FUNCTION_BLOCK I_RPTO (* Primary or Rear Power Take off Output Shaft RPTO *)
  (* Standard: ISO 11783-7; Classification: PGN 65091; Function: Primary or Rear Power Take off Output Shaft RPTO; Description: Copyright (c) 2024 HR Agrartechnik GmbH This program and the accompanying materials are made available under the terms of the Eclipse Public License 2.0 which is available at https://www.eclipse.org/legal/epl-2.0/ SPDX-License-Identifier: EPL-2.0 Message that provides the measurement of the current primary or rear power take-off (PTO) output shaft parameters. https://docs.ms-muc-docs.de/projects/isobus-other-docs/de/latest/PGN/PGN_65091.html *)
  (* Version 1.0, 2024-07-09, Franz Höpfinger, HR Agrartechnik GmbH *)
  PACKAGE isobus::tecu;
  (* Documentation:
  Primary or Rear Power Take off Output Shaft RPTO
   TIMEOUT / IND Vertrag: TIMEOUT feuert ausschliesslich beim tatsaechlichen Eintreten eines Timeouts (Q_timeout wird true). Das Zuruecksetzen von Q_timeout auf false (Timeout vorbei) wird bewusst NICHT nochmal separat ueber TIMEOUT gemeldet, sondern kommt ueber IND - das feuert bei jedem Zyklus ohne aktiven Timeout und publiziert Q_timeout mit. Nachgeschaltete Bausteine, die auf das Ende eines Timeouts reagieren muessen, werten dafuer IND mit Q_timeout==false aus, nicht ein zweites TIMEOUT-Event.
  *)
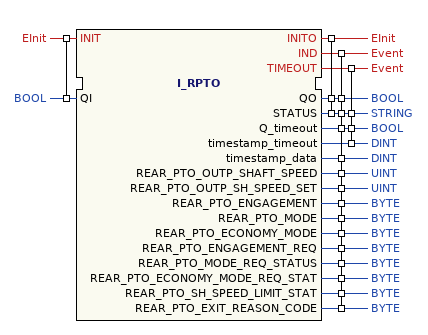
  EVENT_INPUT
    INIT : EInit WITH QI; (* Service Initialization *)
  END_EVENT
  EVENT_OUTPUT
    INITO : EInit WITH QO, STATUS; (* Initialization Confirm *)
    IND WITH QO, timestamp_data, STATUS, Q_timeout, REAR_PTO_OUTP_SHAFT_SPEED, REAR_PTO_OUTP_SH_SPEED_SET, REAR_PTO_ENGAGEMENT, REAR_PTO_MODE, REAR_PTO_ECONOMY_MODE, REAR_PTO_ENGAGEMENT_REQ, REAR_PTO_MODE_REQ_STATUS, REAR_PTO_ECONOMY_MODE_REQ_STAT, REAR_PTO_SH_SPEED_LIMIT_STAT, REAR_PTO_EXIT_REASON_CODE; (* Indication from Resource - feuert bei jedem Zyklus ohne aktiven Timeout und publiziert dabei auch den Reset von Q_timeout auf false. *)
    TIMEOUT WITH timestamp_timeout, STATUS, Q_timeout; (* Feuert ausschliesslich beim tatsaechlichen Eintreten eines Timeouts (Entry-Trigger). Das Zuruecksetzen von Q_timeout auf false wird NICHT hier, sondern ueber IND gemeldet. *)
  END_EVENT
  VAR_INPUT
    QI : BOOL; (* Event Input Qualifier *)
  END_VAR
  VAR_OUTPUT
    QO : BOOL; (* Event Output Qualifier *)
    STATUS : STRING;
    Q_timeout : BOOL;
    timestamp_timeout : DINT;
    timestamp_data : DINT;
    REAR_PTO_OUTP_SHAFT_SPEED : UINT := UINT#16#FFFF; (* Rear PTO output shaft speed (see Attributes for Details) *) {SET_ATTRIBUTE(SPN, 1883)} {SET_ATTRIBUTE(SPN_Name, 'Rear PTO output shaft speed')} {SET_ATTRIBUTE(SP_Position_In_PG, '1-2')} {SET_ATTRIBUTE(SP_Length, 16)} (* 16 bits *) {SET_ATTRIBUTE(Scaling, '0.125 1/min/bit')} {SET_ATTRIBUTE(Offset, )} {SET_ATTRIBUTE(Link, 'https://docs.ms-muc-docs.de/projects/isobus-other-docs/de/latest/PGN/PGN_65091.html#spn-1883-rear-pto-output-shaft-speed')}
    REAR_PTO_OUTP_SH_SPEED_SET : UINT := UINT#16#FFFF; (* Rear PTO Output Shaft Speed Set Point (see Attributes for Details) *) {SET_ATTRIBUTE(SPN, 1885)} {SET_ATTRIBUTE(SPN_Name, 'Rear PTO Output Shaft Speed Set Point')} {SET_ATTRIBUTE(SP_Position_In_PG, '3-4')} {SET_ATTRIBUTE(SP_Length, 16)} (* 16 bits *) {SET_ATTRIBUTE(Scaling, '0.125 1/min/bit')} {SET_ATTRIBUTE(Offset, )} {SET_ATTRIBUTE(Link, 'https://docs.ms-muc-docs.de/projects/isobus-other-docs/de/latest/PGN/PGN_65091.html#spn-1885-rear-pto-output-shaft-speed-set-point')}
    REAR_PTO_ENGAGEMENT : BYTE := BYTE#16#FF; (* Rear Power Take Off Engagement (see Attributes for Details) *) {SET_ATTRIBUTE(SPN, 2408)} {SET_ATTRIBUTE(SPN_Name, 'Rear Power Take Off Engagement')} {SET_ATTRIBUTE(SP_Position_In_PG, '5.7')} {SET_ATTRIBUTE(SP_Length, 2)} (* 2 bits *) {SET_ATTRIBUTE(Scaling, '4 states/2 bit')} {SET_ATTRIBUTE(Offset, )} {SET_ATTRIBUTE(Link, 'https://docs.ms-muc-docs.de/projects/isobus-other-docs/de/latest/PGN/PGN_65091.html#spn-2408-rear-power-take-off-engagement')}
    REAR_PTO_MODE : BYTE := BYTE#16#FF; (* Rear Power Take Off Mode (see Attributes for Details) *) {SET_ATTRIBUTE(SPN, 1890)} {SET_ATTRIBUTE(SPN_Name, 'Rear Power Take Off Mode')} {SET_ATTRIBUTE(SP_Position_In_PG, '5.5')} {SET_ATTRIBUTE(SP_Length, 2)} (* 2 bits *) {SET_ATTRIBUTE(Scaling, '4 states/2 bit')} {SET_ATTRIBUTE(Offset, )} {SET_ATTRIBUTE(Link, 'https://docs.ms-muc-docs.de/projects/isobus-other-docs/de/latest/PGN/PGN_65091.html#spn-1890-rear-power-take-off-mode')}
    REAR_PTO_ECONOMY_MODE : BYTE := BYTE#16#FF; (* Rear Power Take Off Economy Mode (see Attributes for Details) *) {SET_ATTRIBUTE(SPN, 1892)} {SET_ATTRIBUTE(SPN_Name, 'Rear Power Take Off Economy Mode')} {SET_ATTRIBUTE(SP_Position_In_PG, '5.3')} {SET_ATTRIBUTE(SP_Length, 2)} (* 2 bits *) {SET_ATTRIBUTE(Scaling, '4 states/2 bit')} {SET_ATTRIBUTE(Offset, )} {SET_ATTRIBUTE(Link, 'https://docs.ms-muc-docs.de/projects/isobus-other-docs/de/latest/PGN/PGN_65091.html#spn-1892-rear-power-take-off-economy-mode')}
    REAR_PTO_ENGAGEMENT_REQ : BYTE := BYTE#16#FF; (* Rear PTO engagement request status (see Attributes for Details) *) {SET_ATTRIBUTE(SPN, 5156)} {SET_ATTRIBUTE(SPN_Name, 'Rear PTO engagement request status')} {SET_ATTRIBUTE(SP_Position_In_PG, '5.1')} {SET_ATTRIBUTE(SP_Length, 2)} (* 2 bits *) {SET_ATTRIBUTE(Scaling, '4 states/2 bit')} {SET_ATTRIBUTE(Offset, )} {SET_ATTRIBUTE(Link, 'https://docs.ms-muc-docs.de/projects/isobus-other-docs/de/latest/PGN/PGN_65091.html#spn-5156-rear-pto-engagement-request-status')}
    REAR_PTO_MODE_REQ_STATUS : BYTE := BYTE#16#FF; (* Rear PTO mode request status (see Attributes for Details) *) {SET_ATTRIBUTE(SPN, 5157)} {SET_ATTRIBUTE(SPN_Name, 'Rear PTO mode request status')} {SET_ATTRIBUTE(SP_Position_In_PG, '6.7')} {SET_ATTRIBUTE(SP_Length, 2)} (* 2 bits *) {SET_ATTRIBUTE(Scaling, '4 states/2 bit')} {SET_ATTRIBUTE(Offset, )} {SET_ATTRIBUTE(Link, 'https://docs.ms-muc-docs.de/projects/isobus-other-docs/de/latest/PGN/PGN_65091.html#spn-5157-rear-pto-mode-request-status')}
    REAR_PTO_ECONOMY_MODE_REQ_STAT : BYTE := BYTE#16#FF; (* Rear PTO Economy mode request status (see Attributes for Details) *) {SET_ATTRIBUTE(SPN, 5158)} {SET_ATTRIBUTE(SPN_Name, 'Rear PTO Economy mode request status')} {SET_ATTRIBUTE(SP_Position_In_PG, '6.5')} {SET_ATTRIBUTE(SP_Length, 2)} (* 2 bits *) {SET_ATTRIBUTE(Scaling, '4 states/2 bit')} {SET_ATTRIBUTE(Offset, )} {SET_ATTRIBUTE(Link, 'https://docs.ms-muc-docs.de/projects/isobus-other-docs/de/latest/PGN/PGN_65091.html#spn-5158-rear-pto-economy-mode-request-status')}
    REAR_PTO_SH_SPEED_LIMIT_STAT : BYTE := BYTE#16#FF; (* Rear PTO shaft speed limit status (see Attributes for Details) *) {SET_ATTRIBUTE(SPN, 5159)} {SET_ATTRIBUTE(SPN_Name, 'Rear PTO shaft speed limit status')} {SET_ATTRIBUTE(SP_Position_In_PG, '6.2')} {SET_ATTRIBUTE(SP_Length, 3)} (* 3 bits *) {SET_ATTRIBUTE(Scaling, '8 states/3 bit')} {SET_ATTRIBUTE(Offset, )} {SET_ATTRIBUTE(Link, 'https://docs.ms-muc-docs.de/projects/isobus-other-docs/de/latest/PGN/PGN_65091.html#spn-5159-rear-pto-shaft-speed-limit-status')}
    REAR_PTO_EXIT_REASON_CODE : BYTE := BYTE#16#FF; (* Rear PTO exit/reason code (see Attributes for Details) *) {SET_ATTRIBUTE(SPN, 5820)} {SET_ATTRIBUTE(SPN_Name, 'Rear PTO exit/reason code')} {SET_ATTRIBUTE(SP_Position_In_PG, '7.1')} {SET_ATTRIBUTE(SP_Length, 6)} (* 6 bits *) {SET_ATTRIBUTE(Scaling, '64 states/6 bit')} {SET_ATTRIBUTE(Offset, )} {SET_ATTRIBUTE(Link, 'https://docs.ms-muc-docs.de/projects/isobus-other-docs/de/latest/PGN/PGN_65091.html#spn-5820-rear-pto-exit-reason-code')}
  END_VAR
END_FUNCTION_BLOCK
